{attribute 'no_explicit_call' := 'do not call this function block directly'} 
FUNCTION_BLOCK AdsCommunicationSettings EXTENDS CommunicationSettings
VAR_INPUT
	AmsNetId : Tc2_System.T_AmsNetID;
	AmsPort : Tc2_System.T_AmsPort := 801;
END_VAR
VAR
	_ClassName : STRING := __POUNAME();
END_VAR

PROPERTY CommunicationTypeName : STRING
GET
CommunicationTypeName := 'ADS';
END_GET
END_PROPERTY

END_FUNCTION_BLOCK

(* stored: Version 1.1.0.1
   POU AdsCommunicationSettings: Id {f50f2a7b-2d08-499c-8ef2-1045c55b0877}, SpecialFunc None
   Property CommunicationTypeName: Id {9f96a142-d6b3-4118-ab39-4513b798eb92}
   Get Get: Id {c3a73631-212d-4d57-bed9-2c918ac59feb} *)
